PROGRAM UDP

VAR_INPUT
	x	  AT%Q*	: ARRAY[1..4] OF LREAL;
	y	  AT%Q*	: ARRAY[1..4] OF LREAL;
	theta AT%Q*	: ARRAY[1..4] OF LREAL;
END_VAR

VAR
	udp1 : UDPConnect;
	count :INT :=0;
END_VAR

(*** UDP Kommunikation ***
	Hier wird nur der FB UDPConnect instanziert
	Für x,y,theta reichen eigentlich 8 Byte Variablen. Hier: LREAL wegen Kompatibilität
		zu Simulink Regler, der double (=LREAL) als Input braucht
*)

udp1();

END_PROGRAM

(* stored: Version 1.1.0.1, ProductVersion 3.1.4022.3
   POU UDP: Id {0609bed4-bf8f-4f82-907f-a18d61afa454}, SpecialFunc None *)
